// Mitsubishi GX Works2 project: 11-06-2020 Counter_300pulses   PLC: FX3G

PROGRAM MAIN
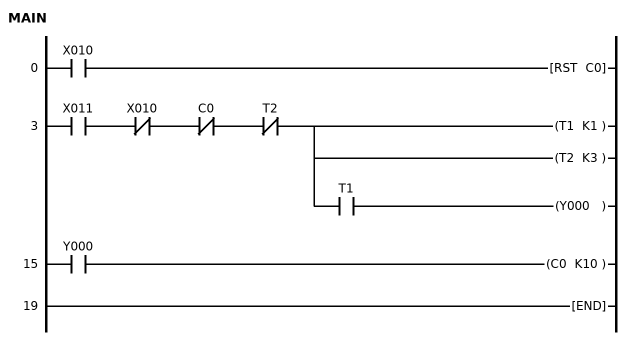
0     LD      X010
      RST     C0
3     LD      X011
      ANI     X010
      ANI     C0
      ANI     T2
      OUT     T1 K1
      OUT     T2 K3
      AND     T1
      OUT     Y000
15    LD      Y000
      OUT     C0 K10
19    END
END_PROGRAM
